	RoomTemp_217: FB_BACnetRM_AI := (Client:=Client,nObjectInstance:=55561);
	TempAdjust_217: FB_BACnetRM_AV := (Client:=Client,nObjectInstance:=55562);
	FilterSign_217: FB_BACnetRM_BI := (Client:=Client,nObjectInstance:=55563);
	FilterSignReset_217: FB_BACnetRM_BV := (Client:=Client,nObjectInstance:=55564);
	RemoteControlStart_217: FB_BACnetRM_BV := (Client:=Client,nObjectInstance:=55565);
	
	RemoteControlTempAdjust_217: FB_BACnetRM_BV := (Client:=Client,nObjectInstance:=55568);
	
	
	
	
	
	
	
	
	
	
	
	
	StartStopCommand_218: FB_BACnetRM_BO := (Client:=Client,nObjectInstance:=55809);
	StartStopStatus_218: FB_BACnetRM_BI := (Client:=Client,nObjectInstance:=55810);
	Alarm_218: FB_BACnetRM_BI := (Client:=Client,nObjectInstance:=55811);
	MalfunctionCode_218: FB_BACnetRM_MI := (Client:=Client,nObjectInstance:=55812);
	
	
	
	
	RoomTemp_218: FB_BACnetRM_AI := (Client:=Client,nObjectInstance:=55817);
	TempAdjust_218: FB_BACnetRM_AV := (Client:=Client,nObjectInstance:=55818);
	FilterSign_218: FB_BACnetRM_BI := (Client:=Client,nObjectInstance:=55819);
	FilterSignReset_218: FB_BACnetRM_BV := (Client:=Client,nObjectInstance:=55820);
	RemoteControlStart_218: FB_BACnetRM_BV := (Client:=Client,nObjectInstance:=55821);
	
	RemoteControlTempAdjust_218: FB_BACnetRM_BV := (Client:=Client,nObjectInstance:=55824);
	
	
	
	
	
	
	
	
	
	
	
	
	StartStopCommand_219: FB_BACnetRM_BO := (Client:=Client,nObjectInstance:=56065);
	StartStopStatus_219: FB_BACnetRM_BI := (Client:=Client,nObjectInstance:=56066);
	Alarm_219: FB_BACnetRM_BI := (Client:=Client,nObjectInstance:=56067);
	MalfunctionCode_219: FB_BACnetRM_MI := (Client:=Client,nObjectInstance:=56068);
	
	
	
	
	RoomTemp_219: FB_BACnetRM_AI := (Client:=Client,nObjectInstance:=56073);
	TempAdjust_219: FB_BACnetRM_AV := (Client:=Client,nObjectInstance:=56074);
	FilterSign_219: FB_BACnetRM_BI := (Client:=Client,nObjectInstance:=56075);
	FilterSignReset_219: FB_BACnetRM_BV := (Client:=Client,nObjectInstance:=56076);
	RemoteControlStart_219: FB_BACnetRM_BV := (Client:=Client,nObjectInstance:=56077);
	
	RemoteControlTempAdjust_219: FB_BACnetRM_BV := (Client:=Client,nObjectInstance:=56080);
	
	
	
	
	
	
	
	
	
	
	
	
	StartStopCommand_220: FB_BACnetRM_BO := (Client:=Client,nObjectInstance:=56321);
	StartStopStatus_220: FB_BACnetRM_BI := (Client:=Client,nObjectInstance:=56322);
	Alarm_220: FB_BACnetRM_BI := (Client:=Client,nObjectInstance:=56323);
	MalfunctionCode_220: FB_BACnetRM_MI := (Client:=Client,nObjectInstance:=56324);
	
	
	
	
	RoomTemp_220: FB_BACnetRM_AI := (Client:=Client,nObjectInstance:=56329);
	TempAdjust_220: FB_BACnetRM_AV := (Client:=Client,nObjectInstance:=56330);
	FilterSign_220: FB_BACnetRM_BI := (Client:=Client,nObjectInstance:=56331);
	FilterSignReset_220: FB_BACnetRM_BV := (Client:=Client,nObjectInstance:=56332);
	RemoteControlStart_220: FB_BACnetRM_BV := (Client:=Client,nObjectInstance:=56333);
	
	RemoteControlTempAdjust_220: FB_BACnetRM_BV := (Client:=Client,nObjectInstance:=56336);
	
	
	
	
	
	
	
	
	
	
	
	
	StartStopCommand_221: FB_BACnetRM_BO := (Client:=Client,nObjectInstance:=56577);
	StartStopStatus_221: FB_BACnetRM_BI := (Client:=Client,nObjectInstance:=56578);
	Alarm_221: FB_BACnetRM_BI := (Client:=Client,nObjectInstance:=56579);
	MalfunctionCode_221: FB_BACnetRM_MI := (Client:=Client,nObjectInstance:=56580);
	
	
	
	
	RoomTemp_221: FB_BACnetRM_AI := (Client:=Client,nObjectInstance:=56585);
	TempAdjust_221: FB_BACnetRM_AV := (Client:=Client,nObjectInstance:=56586);
	FilterSign_221: FB_BACnetRM_BI := (Client:=Client,nObjectInstance:=56587);
	FilterSignReset_221: FB_BACnetRM_BV := (Client:=Client,nObjectInstance:=56588);
	RemoteControlStart_221: FB_BACnetRM_BV := (Client:=Client,nObjectInstance:=56589);
	
	RemoteControlTempAdjust_221: FB_BACnetRM_BV := (Client:=Client,nObjectInstance:=56592);
	
	
	
	
	
	
	
	
	
	
	
	
	StartStopCommand_222: FB_BACnetRM_BO := (Client:=Client,nObjectInstance:=56833);
	StartStopStatus_222: FB_BACnetRM_BI := (Client:=Client,nObjectInstance:=56834);
	Alarm_222: FB_BACnetRM_BI := (Client:=Client,nObjectInstance:=56835);
	MalfunctionCode_222: FB_BACnetRM_MI := (Client:=Client,nObjectInstance:=56836);
	
	
	
	
	RoomTemp_222: FB_BACnetRM_AI := (Client:=Client,nObjectInstance:=56841);
	TempAdjust_222: FB_BACnetRM_AV := (Client:=Client,nObjectInstance:=56842);
	FilterSign_222: FB_BACnetRM_BI := (Client:=Client,nObjectInstance:=56843);
	FilterSignReset_222: FB_BACnetRM_BV := (Client:=Client,nObjectInstance:=56844);
	RemoteControlStart_222: FB_BACnetRM_BV := (Client:=Client,nObjectInstance:=56845);
	
	RemoteControlTempAdjust_222: FB_BACnetRM_BV := (Client:=Client,nObjectInstance:=56848);
	
	
	
	
	
	
	
	
	
	
	
	
	StartStopCommand_223: FB_BACnetRM_BO := (Client:=Client,nObjectInstance:=57089);
	StartStopStatus_223: FB_BACnetRM_BI := (Client:=Client,nObjectInstance:=57090);
	Alarm_223: FB_BACnetRM_BI := (Client:=Client,nObjectInstance:=57091);
	MalfunctionCode_223: FB_BACnetRM_MI := (Client:=Client,nObjectInstance:=57092);
	
	
	
	
	RoomTemp_223: FB_BACnetRM_AI := (Client:=Client,nObjectInstance:=57097);
	TempAdjust_223: FB_BACnetRM_AV := (Client:=Client,nObjectInstance:=57098);
	FilterSign_223: FB_BACnetRM_BI := (Client:=Client,nObjectInstance:=57099);
	FilterSignReset_223: FB_BACnetRM_BV := (Client:=Client,nObjectInstance:=57100);
	RemoteControlStart_223: FB_BACnetRM_BV := (Client:=Client,nObjectInstance:=57101);
	
	RemoteControlTempAdjust_223: FB_BACnetRM_BV := (Client:=Client,nObjectInstance:=57104);
	
	
	
	
	
	
	
	
	
	
	
	
	StartStopCommand_224: FB_BACnetRM_BO := (Client:=Client,nObjectInstance:=57345);
	StartStopStatus_224: FB_BACnetRM_BI := (Client:=Client,nObjectInstance:=57346);
	Alarm_224: FB_BACnetRM_BI := (Client:=Client,nObjectInstance:=57347);
	MalfunctionCode_224: FB_BACnetRM_MI := (Client:=Client,nObjectInstance:=57348);
	
	
	
	
	RoomTemp_224: FB_BACnetRM_AI := (Client:=Client,nObjectInstance:=57353);
	TempAdjust_224: FB_BACnetRM_AV := (Client:=Client,nObjectInstance:=57354);
	FilterSign_224: FB_BACnetRM_BI := (Client:=Client,nObjectInstance:=57355);
	FilterSignReset_224: FB_BACnetRM_BV := (Client:=Client,nObjectInstance:=57356);
	RemoteControlStart_224: FB_BACnetRM_BV := (Client:=Client,nObjectInstance:=57357);
	
	RemoteControlTempAdjust_224: FB_BACnetRM_BV := (Client:=Client,nObjectInstance:=57360);
	
	
	
	
	
	
	
	
	
	
	
	
	StartStopCommand_225: FB_BACnetRM_BO := (Client:=Client,nObjectInstance:=57601);
	StartStopStatus_225: FB_BACnetRM_BI := (Client:=Client,nObjectInstance:=57602);
	Alarm_225: FB_BACnetRM_BI := (Client:=Client,nObjectInstance:=57603);
	MalfunctionCode_225: FB_BACnetRM_MI := (Client:=Client,nObjectInstance:=57604);
	
	
	
	
	RoomTemp_225: FB_BACnetRM_AI := (Client:=Client,nObjectInstance:=57609);
	TempAdjust_225: FB_BACnetRM_AV := (Client:=Client,nObjectInstance:=57610);
	FilterSign_225: FB_BACnetRM_BI := (Client:=Client,nObjectInstance:=57611);
	FilterSignReset_225: FB_BACnetRM_BV := (Client:=Client,nObjectInstance:=57612);
	RemoteControlStart_225: FB_BACnetRM_BV := (Client:=Client,nObjectInstance:=57613);
	
	RemoteControlTempAdjust_225: FB_BACnetRM_BV := (Client:=Client,nObjectInstance:=57616);
	
	
	
	
	
	
	
	
	
	
	
	
	StartStopCommand_226: FB_BACnetRM_BO := (Client:=Client,nObjectInstance:=57857);
	StartStopStatus_226: FB_BACnetRM_BI := (Client:=Client,nObjectInstance:=57858);
	Alarm_226: FB_BACnetRM_BI := (Client:=Client,nObjectInstance:=57859);
	MalfunctionCode_226: FB_BACnetRM_MI := (Client:=Client,nObjectInstance:=57860);
	
	
	
	
	RoomTemp_226: FB_BACnetRM_AI := (Client:=Client,nObjectInstance:=57865);
	TempAdjust_226: FB_BACnetRM_AV := (Client:=Client,nObjectInstance:=57866);
	FilterSign_226: FB_BACnetRM_BI := (Client:=Client,nObjectInstance:=57867);
	FilterSignReset_226: FB_BACnetRM_BV := (Client:=Client,nObjectInstance:=57868);
	RemoteControlStart_226: FB_BACnetRM_BV := (Client:=Client,nObjectInstance:=57869);
	
	RemoteControlTempAdjust_226: FB_BACnetRM_BV := (Client:=Client,nObjectInstance:=57872);
	
	
	
	
	
	
	
	
	
	
	
	
	StartStopCommand_227: FB_BACnetRM_BO := (Client:=Client,nObjectInstance:=58113);
	StartStopStatus_227: FB_BACnetRM_BI := (Client:=Client,nObjectInstance:=58114);
	Alarm_227: FB_BACnetRM_BI := (Client:=Client,nObjectInstance:=58115);
	MalfunctionCode_227: FB_BACnetRM_MI := (Client:=Client,nObjectInstance:=58116);
	
	
	
	
	RoomTemp_227: FB_BACnetRM_AI := (Client:=Client,nObjectInstance:=58121);
	TempAdjust_227: FB_BACnetRM_AV := (Client:=Client,nObjectInstance:=58122);
	FilterSign_227: FB_BACnetRM_BI := (Client:=Client,nObjectInstance:=58123);
	FilterSignReset_227: FB_BACnetRM_BV := (Client:=Client,nObjectInstance:=58124);
	RemoteControlStart_227: FB_BACnetRM_BV := (Client:=Client,nObjectInstance:=58125);
	
	RemoteControlTempAdjust_227: FB_BACnetRM_BV := (Client:=Client,nObjectInstance:=58128);
	
	
	
	
	
	
	
	
	
	
	
	
	StartStopCommand_228: FB_BACnetRM_BO := (Client:=Client,nObjectInstance:=58369);
	StartStopStatus_228: FB_BACnetRM_BI := (Client:=Client,nObjectInstance:=58370);
	Alarm_228: FB_BACnetRM_BI := (Client:=Client,nObjectInstance:=58371);
	MalfunctionCode_228: FB_BACnetRM_MI := (Client:=Client,nObjectInstance:=58372);
	
	
	
	
	RoomTemp_228: FB_BACnetRM_AI := (Client:=Client,nObjectInstance:=58377);
	TempAdjust_228: FB_BACnetRM_AV := (Client:=Client,nObjectInstance:=58378);
	FilterSign_228: FB_BACnetRM_BI := (Client:=Client,nObjectInstance:=58379);
	FilterSignReset_228: FB_BACnetRM_BV := (Client:=Client,nObjectInstance:=58380);
	RemoteControlStart_228: FB_BACnetRM_BV := (Client:=Client,nObjectInstance:=58381);
	
	RemoteControlTempAdjust_228: FB_BACnetRM_BV := (Client:=Client,nObjectInstance:=58384);
	
	
	
	
	
	
	
	
	
	
	
	
	StartStopCommand_229: FB_BACnetRM_BO := (Client:=Client,nObjectInstance:=58625);
	StartStopStatus_229: FB_BACnetRM_BI := (Client:=Client,nObjectInstance:=58626);
	Alarm_229: FB_BACnetRM_BI := (Client:=Client,nObjectInstance:=58627);
	MalfunctionCode_229: FB_BACnetRM_MI := (Client:=Client,nObjectInstance:=58628);
	
	
	
	
	RoomTemp_229: FB_BACnetRM_AI := (Client:=Client,nObjectInstance:=58633);
	TempAdjust_229: FB_BACnetRM_AV := (Client:=Client,nObjectInstance:=58634);
	FilterSign_229: FB_BACnetRM_BI := (Client:=Client,nObjectInstance:=58635);
	FilterSignReset_229: FB_BACnetRM_BV := (Client:=Client,nObjectInstance:=58636);
	RemoteControlStart_229: FB_BACnetRM_BV := (Client:=Client,nObjectInstance:=58637);
	
	RemoteControlTempAdjust_229: FB_BACnetRM_BV := (Client:=Client,nObjectInstance:=58640);
	
	
	
	
	
	
	
	
	
	
	
	
	StartStopCommand_230: FB_BACnetRM_BO := (Client:=Client,nObjectInstance:=58881);
	StartStopStatus_230: FB_BACnetRM_BI := (Client:=Client,nObjectInstance:=58882);
	Alarm_230: FB_BACnetRM_BI := (Client:=Client,nObjectInstance:=58883);
	MalfunctionCode_230: FB_BACnetRM_MI := (Client:=Client,nObjectInstance:=58884);
	
	
	
	
	RoomTemp_230: FB_BACnetRM_AI := (Client:=Client,nObjectInstance:=58889);
	TempAdjust_230: FB_BACnetRM_AV := (Client:=Client,nObjectInstance:=58890);
	FilterSign_230: FB_BACnetRM_BI := (Client:=Client,nObjectInstance:=58891);
	FilterSignReset_230: FB_BACnetRM_BV := (Client:=Client,nObjectInstance:=58892);
	RemoteControlStart_230: FB_BACnetRM_BV := (Client:=Client,nObjectInstance:=58893);
	
	RemoteControlTempAdjust_230: FB_BACnetRM_BV := (Client:=Client,nObjectInstance:=58896);
	
	
	
	
	
	
	
	
	
	
	
	
	StartStopCommand_231: FB_BACnetRM_BO := (Client:=Client,nObjectInstance:=59137);
	StartStopStatus_231: FB_BACnetRM_BI := (Client:=Client,nObjectInstance:=59138);
	Alarm_231: FB_BACnetRM_BI := (Client:=Client,nObjectInstance:=59139);
	MalfunctionCode_231: FB_BACnetRM_MI := (Client:=Client,nObjectInstance:=59140);
	
	
	
	
	RoomTemp_231: FB_BACnetRM_AI := (Client:=Client,nObjectInstance:=59145);
	TempAdjust_231: FB_BACnetRM_AV := (Client:=Client,nObjectInstance:=59146);
	FilterSign_231: FB_BACnetRM_BI := (Client:=Client,nObjectInstance:=59147);
	FilterSignReset_231: FB_BACnetRM_BV := (Client:=Client,nObjectInstance:=59148);
	RemoteControlStart_231: FB_BACnetRM_BV := (Client:=Client,nObjectInstance:=59149);
	
	RemoteControlTempAdjust_231: FB_BACnetRM_BV := (Client:=Client,nObjectInstance:=59152);
	
	
	
	
	
	
	
	
	
	
	
	
	StartStopCommand_232: FB_BACnetRM_BO := (Client:=Client,nObjectInstance:=59393);
	StartStopStatus_232: FB_BACnetRM_BI := (Client:=Client,nObjectInstance:=59394);
	Alarm_232: FB_BACnetRM_BI := (Client:=Client,nObjectInstance:=59395);
	MalfunctionCode_232: FB_BACnetRM_MI := (Client:=Client,nObjectInstance:=59396);
	
	
	
	
	RoomTemp_232: FB_BACnetRM_AI := (Client:=Client,nObjectInstance:=59401);
	TempAdjust_232: FB_BACnetRM_AV := (Client:=Client,nObjectInstance:=59402);
	FilterSign_232: FB_BACnetRM_BI := (Client:=Client,nObjectInstance:=59403);
	FilterSignReset_232: FB_BACnetRM_BV := (Client:=Client,nObjectInstance:=59404);
	RemoteControlStart_232: FB_BACnetRM_BV := (Client:=Client,nObjectInstance:=59405);
	
	RemoteControlTempAdjust_232: FB_BACnetRM_BV := (Client:=Client,nObjectInstance:=59408);
	
	
	
	
	
	
	
	
	
	
	
	
	StartStopCommand_233: FB_BACnetRM_BO := (Client:=Client,nObjectInstance:=59649);
	StartStopStatus_233: FB_BACnetRM_BI := (Client:=Client,nObjectInstance:=59650);
	Alarm_233: FB_BACnetRM_BI := (Client:=Client,nObjectInstance:=59651);
	MalfunctionCode_233: FB_BACnetRM_MI := (Client:=Client,nObjectInstance:=59652);
	
	
	
	
	RoomTemp_233: FB_BACnetRM_AI := (Client:=Client,nObjectInstance:=59657);
	TempAdjust_233: FB_BACnetRM_AV := (Client:=Client,nObjectInstance:=59658);
	FilterSign_233: FB_BACnetRM_BI := (Client:=Client,nObjectInstance:=59659);
	FilterSignReset_233: FB_BACnetRM_BV := (Client:=Client,nObjectInstance:=59660);
	RemoteControlStart_233: FB_BACnetRM_BV := (Client:=Client,nObjectInstance:=59661);
	
	RemoteControlTempAdjust_233: FB_BACnetRM_BV := (Client:=Client,nObjectInstance:=59664);
	
	
	
	
	
	
	
	
	
	
	
	
	StartStopCommand_234: FB_BACnetRM_BO := (Client:=Client,nObjectInstance:=59905);
	StartStopStatus_234: FB_BACnetRM_BI := (Client:=Client,nObjectInstance:=59906);
	Alarm_234: FB_BACnetRM_BI := (Client:=Client,nObjectInstance:=59907);
	MalfunctionCode_234: FB_BACnetRM_MI := (Client:=Client,nObjectInstance:=59908);
	
	
	
	
	RoomTemp_234: FB_BACnetRM_AI := (Client:=Client,nObjectInstance:=59913);
	TempAdjust_234: FB_BACnetRM_AV := (Client:=Client,nObjectInstance:=59914);
	FilterSign_234: FB_BACnetRM_BI := (Client:=Client,nObjectInstance:=59915);
	FilterSignReset_234: FB_BACnetRM_BV := (Client:=Client,nObjectInstance:=59916);
	RemoteControlStart_234: FB_BACnetRM_BV := (Client:=Client,nObjectInstance:=59917);
	
	RemoteControlTempAdjust_234: FB_BACnetRM_BV := (Client:=Client,nObjectInstance:=59920);
	
	
	
	
	
	
	
	
	
	
	
	
	StartStopCommand_235: FB_BACnetRM_BO := (Client:=Client,nObjectInstance:=60161);
	StartStopStatus_235: FB_BACnetRM_BI := (Client:=Client,nObjectInstance:=60162);
	Alarm_235: FB_BACnetRM_BI := (Client:=Client,nObjectInstance:=60163);
	MalfunctionCode_235: FB_BACnetRM_MI := (Client:=Client,nObjectInstance:=60164);
	
	
	
	
	RoomTemp_235: FB_BACnetRM_AI := (Client:=Client,nObjectInstance:=60169);
	TempAdjust_235: FB_BACnetRM_AV := (Client:=Client,nObjectInstance:=60170);
	FilterSign_235: FB_BACnetRM_BI := (Client:=Client,nObjectInstance:=60171);
	FilterSignReset_235: FB_BACnetRM_BV := (Client:=Client,nObjectInstance:=60172);
	RemoteControlStart_235: FB_BACnetRM_BV := (Client:=Client,nObjectInstance:=60173);
	
	RemoteControlTempAdjust_235: FB_BACnetRM_BV := (Client:=Client,nObjectInstance:=60176);
	
	
	
	
	
	
	
	
	
	
	
	
	StartStopCommand_236: FB_BACnetRM_BO := (Client:=Client,nObjectInstance:=60417);
	StartStopStatus_236: FB_BACnetRM_BI := (Client:=Client,nObjectInstance:=60418);
	Alarm_236: FB_BACnetRM_BI := (Client:=Client,nObjectInstance:=60419);
	MalfunctionCode_236: FB_BACnetRM_MI := (Client:=Client,nObjectInstance:=60420);
	
	
	
	
	RoomTemp_236: FB_BACnetRM_AI := (Client:=Client,nObjectInstance:=60425);
	TempAdjust_236: FB_BACnetRM_AV := (Client:=Client,nObjectInstance:=60426);
	FilterSign_236: FB_BACnetRM_BI := (Client:=Client,nObjectInstance:=60427);
	FilterSignReset_236: FB_BACnetRM_BV := (Client:=Client,nObjectInstance:=60428);
	RemoteControlStart_236: FB_BACnetRM_BV := (Client:=Client,nObjectInstance:=60429);
	
	RemoteControlTempAdjust_236: FB_BACnetRM_BV := (Client:=Client,nObjectInstance:=60432);
	
	
	
	
	
	
	
	
	
	
	
	
	StartStopCommand_237: FB_BACnetRM_BO := (Client:=Client,nObjectInstance:=60673);
	StartStopStatus_237: FB_BACnetRM_BI := (Client:=Client,nObjectInstance:=60674);
	Alarm_237: FB_BACnetRM_BI := (Client:=Client,nObjectInstance:=60675);
	MalfunctionCode_237: FB_BACnetRM_MI := (Client:=Client,nObjectInstance:=60676);
	
	
	
	
	RoomTemp_237: FB_BACnetRM_AI := (Client:=Client,nObjectInstance:=60681);
	TempAdjust_237: FB_BACnetRM_AV := (Client:=Client,nObjectInstance:=60682);
	FilterSign_237: FB_BACnetRM_BI := (Client:=Client,nObjectInstance:=60683);
	FilterSignReset_237: FB_BACnetRM_BV := (Client:=Client,nObjectInstance:=60684);
	RemoteControlStart_237: FB_BACnetRM_BV := (Client:=Client,nObjectInstance:=60685);
	
	RemoteControlTempAdjust_237: FB_BACnetRM_BV := (Client:=Client,nObjectInstance:=60688);
	
	
	
	
	
	
	
	
	
	
	
	
	StartStopCommand_238: FB_BACnetRM_BO := (Client:=Client,nObjectInstance:=60929);
	StartStopStatus_238: FB_BACnetRM_BI := (Client:=Client,nObjectInstance:=60930);
	Alarm_238: FB_BACnetRM_BI := (Client:=Client,nObjectInstance:=60931);
	MalfunctionCode_238: FB_BACnetRM_MI := (Client:=Client,nObjectInstance:=60932);
	
	
	
	
	RoomTemp_238: FB_BACnetRM_AI := (Client:=Client,nObjectInstance:=60937);
	TempAdjust_238: FB_BACnetRM_AV := (Client:=Client,nObjectInstance:=60938);
	FilterSign_238: FB_BACnetRM_BI := (Client:=Client,nObjectInstance:=60939);
	FilterSignReset_238: FB_BACnetRM_BV := (Client:=Client,nObjectInstance:=60940);
	RemoteControlStart_238: FB_BACnetRM_BV := (Client:=Client,nObjectInstance:=60941);
	
	RemoteControlTempAdjust_238: FB_BACnetRM_BV := (Client:=Client,nObjectInstance:=60944);
	
	
	
	
	
	
	
	
	
	
	
	
	StartStopCommand_241: FB_BACnetRM_BO := (Client:=Client,nObjectInstance:=61697);
	StartStopStatus_241: FB_BACnetRM_BI := (Client:=Client,nObjectInstance:=61698);
	Alarm_241: FB_BACnetRM_BI := (Client:=Client,nObjectInstance:=61699);
	MalfunctionCode_241: FB_BACnetRM_MI := (Client:=Client,nObjectInstance:=61700);
	
	
	
	
	RoomTemp_241: FB_BACnetRM_AI := (Client:=Client,nObjectInstance:=61705);
	TempAdjust_241: FB_BACnetRM_AV := (Client:=Client,nObjectInstance:=61706);
	FilterSign_241: FB_BACnetRM_BI := (Client:=Client,nObjectInstance:=61707);
	FilterSignReset_241: FB_BACnetRM_BV := (Client:=Client,nObjectInstance:=61708);
	RemoteControlStart_241: FB_BACnetRM_BV := (Client:=Client,nObjectInstance:=61709);
	
	RemoteControlTempAdjust_241: FB_BACnetRM_BV := (Client:=Client,nObjectInstance:=61712);
	
	
	
	
	
	
	
	
	
	
	
	
	StartStopCommand_242: FB_BACnetRM_BO := (Client:=Client,nObjectInstance:=61953);
	StartStopStatus_242: FB_BACnetRM_BI := (Client:=Client,nObjectInstance:=61954);
	Alarm_242: FB_BACnetRM_BI := (Client:=Client,nObjectInstance:=61955);
	MalfunctionCode_242: FB_BACnetRM_MI := (Client:=Client,nObjectInstance:=61956);
	
	
	
	
	RoomTemp_242: FB_BACnetRM_AI := (Client:=Client,nObjectInstance:=61961);
	TempAdjust_242: FB_BACnetRM_AV := (Client:=Client,nObjectInstance:=61962);
	FilterSign_242: FB_BACnetRM_BI := (Client:=Client,nObjectInstance:=61963);
	FilterSignReset_242: FB_BACnetRM_BV := (Client:=Client,nObjectInstance:=61964);
	RemoteControlStart_242: FB_BACnetRM_BV := (Client:=Client,nObjectInstance:=61965);
	
	RemoteControlTempAdjust_242: FB_BACnetRM_BV := (Client:=Client,nObjectInstance:=61968);
	
	
	
	
	
	
	
	
	
	
	
	
	StartStopCommand_243: FB_BACnetRM_BO := (Client:=Client,nObjectInstance:=62209);
	StartStopStatus_243: FB_BACnetRM_BI := (Client:=Client,nObjectInstance:=62210);
	Alarm_243: FB_BACnetRM_BI := (Client:=Client,nObjectInstance:=62211);
	MalfunctionCode_243: FB_BACnetRM_MI := (Client:=Client,nObjectInstance:=62212);
	
	
	
	
	RoomTemp_243: FB_BACnetRM_AI := (Client:=Client,nObjectInstance:=62217);
	TempAdjust_243: FB_BACnetRM_AV := (Client:=Client,nObjectInstance:=62218);
	FilterSign_243: FB_BACnetRM_BI := (Client:=Client,nObjectInstance:=62219);
	FilterSignReset_243: FB_BACnetRM_BV := (Client:=Client,nObjectInstance:=62220);
	RemoteControlStart_243: FB_BACnetRM_BV := (Client:=Client,nObjectInstance:=62221);
	
	RemoteControlTempAdjust_243: FB_BACnetRM_BV := (Client:=Client,nObjectInstance:=62224);
	
	
	
	
	
	
	
	
	
	
	
	
	CL_Rejection_000: FB_BACnetRM_BV := (Client:=Client,nObjectInstance:=17);
	SystemForcedOff_000: FB_BACnetRM_BV := (Client:=Client,nObjectInstance:=21);
	CL_Rejection_064: FB_BACnetRM_BV := (Client:=Client,nObjectInstance:=16401);
	SystemForcedOff_064: FB_BACnetRM_BV := (Client:=Client,nObjectInstance:=16405);
	CL_Rejection_128: FB_BACnetRM_BV := (Client:=Client,nObjectInstance:=32785);
	SystemForcedOff_128: FB_BACnetRM_BV := (Client:=Client,nObjectInstance:=32789);
	CL_Rejection_192: FB_BACnetRM_BV := (Client:=Client,nObjectInstance:=49169);
	SystemForcedOff_192: FB_BACnetRM_BV := (Client:=Client,nObjectInstance:=49173);
END_VAR

Client();
DAIKIN_MasterStation_III_No_10();
StartStopCommand_000();
StartStopStatus_000();
Alarm_000();
MalfunctionCode_000();




RoomTemp_000();
TempAdjust_000();
FilterSign_000();
FilterSignReset_000();
RemoteControlStart_000();

RemoteControlTempAdjust_000();












StartStopCommand_001();
StartStopStatus_001();
Alarm_001();
MalfunctionCode_001();




RoomTemp_001();
TempAdjust_001();
FilterSign_001();
FilterSignReset_001();
RemoteControlStart_001();

RemoteControlTempAdjust_001();












StartStopCommand_002();
StartStopStatus_002();
Alarm_002();
MalfunctionCode_002();




RoomTemp_002();
TempAdjust_002();
FilterSign_002();
FilterSignReset_002();
RemoteControlStart_002();

RemoteControlTempAdjust_002();












StartStopCommand_003();
StartStopStatus_003();
Alarm_003();
MalfunctionCode_003();




RoomTemp_003();
TempAdjust_003();
FilterSign_003();
FilterSignReset_003();
RemoteControlStart_003();

RemoteControlTempAdjust_003();












StartStopCommand_004();
StartStopStatus_004();
Alarm_004();
MalfunctionCode_004();




RoomTemp_004();
TempAdjust_004();
FilterSign_004();
FilterSignReset_004();
RemoteControlStart_004();

RemoteControlTempAdjust_004();












StartStopCommand_005();
StartStopStatus_005();
Alarm_005();
MalfunctionCode_005();




RoomTemp_005();
TempAdjust_005();
FilterSign_005();
FilterSignReset_005();
RemoteControlStart_005();

RemoteControlTempAdjust_005();












StartStopCommand_006();
StartStopStatus_006();
Alarm_006();
MalfunctionCode_006();




RoomTemp_006();
TempAdjust_006();
FilterSign_006();
FilterSignReset_006();
RemoteControlStart_006();

RemoteControlTempAdjust_006();












StartStopCommand_007();
StartStopStatus_007();
Alarm_007();
MalfunctionCode_007();




RoomTemp_007();
TempAdjust_007();
FilterSign_007();
FilterSignReset_007();
RemoteControlStart_007();

RemoteControlTempAdjust_007();












StartStopCommand_008();
StartStopStatus_008();
Alarm_008();
MalfunctionCode_008();




RoomTemp_008();
TempAdjust_008();
FilterSign_008();
FilterSignReset_008();
RemoteControlStart_008();

RemoteControlTempAdjust_008();












StartStopCommand_009();
StartStopStatus_009();
Alarm_009();
MalfunctionCode_009();




RoomTemp_009();
TempAdjust_009();
FilterSign_009();
FilterSignReset_009();
RemoteControlStart_009();

RemoteControlTempAdjust_009();












StartStopCommand_010();
StartStopStatus_010();
Alarm_010();
MalfunctionCode_010();




RoomTemp_010();
TempAdjust_010();
FilterSign_010();
FilterSignReset_010();
RemoteControlStart_010();

RemoteControlTempAdjust_010();












StartStopCommand_011();
StartStopStatus_011();
Alarm_011();
MalfunctionCode_011();




RoomTemp_011();
TempAdjust_011();
FilterSign_011();
FilterSignReset_011();
RemoteControlStart_011();

RemoteControlTempAdjust_011();












StartStopCommand_012();
StartStopStatus_012();
Alarm_012();
MalfunctionCode_012();




RoomTemp_012();
TempAdjust_012();
FilterSign_012();
FilterSignReset_012();
RemoteControlStart_012();

RemoteControlTempAdjust_012();












StartStopCommand_013();
StartStopStatus_013();
Alarm_013();
MalfunctionCode_013();




RoomTemp_013();
TempAdjust_013();
FilterSign_013();
FilterSignReset_013();
RemoteControlStart_013();

RemoteControlTempAdjust_013();












StartStopCommand_014();
StartStopStatus_014();
Alarm_014();
MalfunctionCode_014();




RoomTemp_014();
TempAdjust_014();
FilterSign_014();
FilterSignReset_014();
RemoteControlStart_014();

RemoteControlTempAdjust_014();












StartStopCommand_015();
StartStopStatus_015();
Alarm_015();
MalfunctionCode_015();




RoomTemp_015();
TempAdjust_015();
FilterSign_015();
FilterSignReset_015();
RemoteControlStart_015();

RemoteControlTempAdjust_015();












StartStopCommand_016();
StartStopStatus_016();
Alarm_016();
MalfunctionCode_016();




RoomTemp_016();
TempAdjust_016();
FilterSign_016();
FilterSignReset_016();
RemoteControlStart_016();

RemoteControlTempAdjust_016();












StartStopCommand_017();
StartStopStatus_017();
Alarm_017();
MalfunctionCode_017();




RoomTemp_017();
TempAdjust_017();
FilterSign_017();
FilterSignReset_017();
RemoteControlStart_017();

RemoteControlTempAdjust_017();












StartStopCommand_018();
StartStopStatus_018();
Alarm_018();
MalfunctionCode_018();




RoomTemp_018();
TempAdjust_018();
FilterSign_018();
FilterSignReset_018();
RemoteControlStart_018();

RemoteControlTempAdjust_018();












StartStopCommand_019();
StartStopStatus_019();
Alarm_019();
MalfunctionCode_019();




RoomTemp_019();
TempAdjust_019();
FilterSign_019();
FilterSignReset_019();
RemoteControlStart_019();

RemoteControlTempAdjust_019();












StartStopCommand_020();
StartStopStatus_020();
Alarm_020();
MalfunctionCode_020();




RoomTemp_020();
TempAdjust_020();
FilterSign_020();
FilterSignReset_020();
RemoteControlStart_020();

RemoteControlTempAdjust_020();












StartStopCommand_021();
StartStopStatus_021();
Alarm_021();
MalfunctionCode_021();




RoomTemp_021();
TempAdjust_021();
FilterSign_021();
FilterSignReset_021();
RemoteControlStart_021();

RemoteControlTempAdjust_021();












StartStopCommand_048();
StartStopStatus_048();
Alarm_048();
MalfunctionCode_048();




RoomTemp_048();
TempAdjust_048();
FilterSign_048();
FilterSignReset_048();
RemoteControlStart_048();

RemoteControlTempAdjust_048();












StartStopCommand_049();
StartStopStatus_049();
Alarm_049();
MalfunctionCode_049();




RoomTemp_049();
TempAdjust_049();
FilterSign_049();
FilterSignReset_049();
RemoteControlStart_049();

RemoteControlTempAdjust_049();












StartStopCommand_064();
StartStopStatus_064();
Alarm_064();
MalfunctionCode_064();




RoomTemp_064();
TempAdjust_064();
FilterSign_064();
FilterSignReset_064();
RemoteControlStart_064();

RemoteControlTempAdjust_064();












StartStopCommand_065();
StartStopStatus_065();
Alarm_065();
MalfunctionCode_065();




RoomTemp_065();
TempAdjust_065();
FilterSign_065();
FilterSignReset_065();
RemoteControlStart_065();

RemoteControlTempAdjust_065();












StartStopCommand_066();
StartStopStatus_066();
Alarm_066();
MalfunctionCode_066();




RoomTemp_066();
TempAdjust_066();
FilterSign_066();
FilterSignReset_066();
RemoteControlStart_066();

RemoteControlTempAdjust_066();












StartStopCommand_067();
StartStopStatus_067();
Alarm_067();
MalfunctionCode_067();




RoomTemp_067();
TempAdjust_067();
FilterSign_067();
FilterSignReset_067();
RemoteControlStart_067();

RemoteControlTempAdjust_067();












StartStopCommand_068();
StartStopStatus_068();
Alarm_068();
MalfunctionCode_068();




RoomTemp_068();
TempAdjust_068();
FilterSign_068();
FilterSignReset_068();
RemoteControlStart_068();

RemoteControlTempAdjust_068();












StartStopCommand_069();
StartStopStatus_069();
Alarm_069();
MalfunctionCode_069();




RoomTemp_069();
TempAdjust_069();
FilterSign_069();
FilterSignReset_069();
RemoteControlStart_069();

RemoteControlTempAdjust_069();












StartStopCommand_070();
StartStopStatus_070();
Alarm_070();
MalfunctionCode_070();




RoomTemp_070();
TempAdjust_070();
FilterSign_070();
FilterSignReset_070();
RemoteControlStart_070();

RemoteControlTempAdjust_070();












StartStopCommand_071();
StartStopStatus_071();
Alarm_071();
MalfunctionCode_071();




RoomTemp_071();
TempAdjust_071();
FilterSign_071();
FilterSignReset_071();
RemoteControlStart_071();

RemoteControlTempAdjust_071();












StartStopCommand_072();
StartStopStatus_072();
Alarm_072();
MalfunctionCode_072();




RoomTemp_072();
TempAdjust_072();
FilterSign_072();
FilterSignReset_072();
RemoteControlStart_072();

RemoteControlTempAdjust_072();












StartStopCommand_073();
StartStopStatus_073();
Alarm_073();
MalfunctionCode_073();




RoomTemp_073();
TempAdjust_073();
FilterSign_073();
FilterSignReset_073();
RemoteControlStart_073();

RemoteControlTempAdjust_073();












StartStopCommand_074();
StartStopStatus_074();
Alarm_074();
MalfunctionCode_074();




RoomTemp_074();
TempAdjust_074();
FilterSign_074();
FilterSignReset_074();
RemoteControlStart_074();

RemoteControlTempAdjust_074();












StartStopCommand_075();
StartStopStatus_075();
Alarm_075();
MalfunctionCode_075();




RoomTemp_075();
TempAdjust_075();
FilterSign_075();
FilterSignReset_075();
RemoteControlStart_075();

RemoteControlTempAdjust_075();












StartStopCommand_076();
StartStopStatus_076();
Alarm_076();
MalfunctionCode_076();




RoomTemp_076();
TempAdjust_076();
FilterSign_076();
FilterSignReset_076();
RemoteControlStart_076();

RemoteControlTempAdjust_076();












StartStopCommand_077();
StartStopStatus_077();
Alarm_077();
MalfunctionCode_077();




RoomTemp_077();
TempAdjust_077();
FilterSign_077();
FilterSignReset_077();
RemoteControlStart_077();

RemoteControlTempAdjust_077();












StartStopCommand_078();
StartStopStatus_078();
Alarm_078();
MalfunctionCode_078();




RoomTemp_078();
TempAdjust_078();
FilterSign_078();
FilterSignReset_078();
RemoteControlStart_078();

RemoteControlTempAdjust_078();












StartStopCommand_079();
StartStopStatus_079();
Alarm_079();
MalfunctionCode_079();




RoomTemp_079();
TempAdjust_079();
FilterSign_079();
FilterSignReset_079();
RemoteControlStart_079();

RemoteControlTempAdjust_079();












StartStopCommand_080();
StartStopStatus_080();
Alarm_080();
MalfunctionCode_080();




RoomTemp_080();
TempAdjust_080();
FilterSign_080();
FilterSignReset_080();
RemoteControlStart_080();

RemoteControlTempAdjust_080();












StartStopCommand_081();
StartStopStatus_081();
Alarm_081();
MalfunctionCode_081();




RoomTemp_081();
TempAdjust_081();
FilterSign_081();
FilterSignReset_081();
RemoteControlStart_081();

RemoteControlTempAdjust_081();












StartStopCommand_082();
StartStopStatus_082();
Alarm_082();
MalfunctionCode_082();




RoomTemp_082();
TempAdjust_082();
FilterSign_082();
FilterSignReset_082();
RemoteControlStart_082();

RemoteControlTempAdjust_082();












StartStopCommand_083();
StartStopStatus_083();
Alarm_083();
MalfunctionCode_083();




RoomTemp_083();
TempAdjust_083();
FilterSign_083();
FilterSignReset_083();
RemoteControlStart_083();

RemoteControlTempAdjust_083();












StartStopCommand_084();
StartStopStatus_084();
Alarm_084();
MalfunctionCode_084();




RoomTemp_084();
TempAdjust_084();
FilterSign_084();
FilterSignReset_084();
RemoteControlStart_084();

RemoteControlTempAdjust_084();












StartStopCommand_085();
StartStopStatus_085();
Alarm_085();
MalfunctionCode_085();




RoomTemp_085();
TempAdjust_085();
FilterSign_085();
FilterSignReset_085();
RemoteControlStart_085();

RemoteControlTempAdjust_085();












StartStopCommand_096();
StartStopStatus_096();
Alarm_096();
MalfunctionCode_096();




RoomTemp_096();
TempAdjust_096();
FilterSign_096();
FilterSignReset_096();
RemoteControlStart_096();

RemoteControlTempAdjust_096();












StartStopCommand_097();
StartStopStatus_097();
Alarm_097();
MalfunctionCode_097();




RoomTemp_097();
TempAdjust_097();
FilterSign_097();
FilterSignReset_097();
RemoteControlStart_097();

RemoteControlTempAdjust_097();












StartStopCommand_112();
StartStopStatus_112();
Alarm_112();
MalfunctionCode_112();




RoomTemp_112();
TempAdjust_112();
FilterSign_112();
FilterSignReset_112();
RemoteControlStart_112();

RemoteControlTempAdjust_112();












StartStopCommand_128();
StartStopStatus_128();
Alarm_128();
MalfunctionCode_128();




RoomTemp_128();
TempAdjust_128();
FilterSign_128();
FilterSignReset_128();
RemoteControlStart_128();

RemoteControlTempAdjust_128();












StartStopCommand_129();
StartStopStatus_129();
Alarm_129();
MalfunctionCode_129();




RoomTemp_129();
TempAdjust_129();
FilterSign_129();
FilterSignReset_129();
RemoteControlStart_129();

RemoteControlTempAdjust_129();












StartStopCommand_130();
StartStopStatus_130();
Alarm_130();
MalfunctionCode_130();




RoomTemp_130();
TempAdjust_130();
FilterSign_130();
FilterSignReset_130();
RemoteControlStart_130();

RemoteControlTempAdjust_130();












StartStopCommand_131();
StartStopStatus_131();
Alarm_131();
MalfunctionCode_131();




RoomTemp_131();
TempAdjust_131();
FilterSign_131();
FilterSignReset_131();
RemoteControlStart_131();

RemoteControlTempAdjust_131();












StartStopCommand_132();
StartStopStatus_132();
Alarm_132();
MalfunctionCode_132();




RoomTemp_132();
TempAdjust_132();
FilterSign_132();
FilterSignReset_132();
RemoteControlStart_132();

RemoteControlTempAdjust_132();












StartStopCommand_133();
StartStopStatus_133();
Alarm_133();
MalfunctionCode_133();




RoomTemp_133();
TempAdjust_133();
FilterSign_133();
FilterSignReset_133();
RemoteControlStart_133();

RemoteControlTempAdjust_133();












StartStopCommand_134();
StartStopStatus_134();
Alarm_134();
MalfunctionCode_134();




RoomTemp_134();
TempAdjust_134();
FilterSign_134();
FilterSignReset_134();
RemoteControlStart_134();

RemoteControlTempAdjust_134();












StartStopCommand_135();
StartStopStatus_135();
Alarm_135();
MalfunctionCode_135();




RoomTemp_135();
TempAdjust_135();
FilterSign_135();
FilterSignReset_135();
RemoteControlStart_135();

RemoteControlTempAdjust_135();












StartStopCommand_136();
StartStopStatus_136();
Alarm_136();
MalfunctionCode_136();




RoomTemp_136();
TempAdjust_136();
FilterSign_136();
FilterSignReset_136();
RemoteControlStart_136();

RemoteControlTempAdjust_136();












StartStopCommand_137();
StartStopStatus_137();
Alarm_137();
MalfunctionCode_137();




RoomTemp_137();
TempAdjust_137();
FilterSign_137();
FilterSignReset_137();
RemoteControlStart_137();

RemoteControlTempAdjust_137();












StartStopCommand_138();
StartStopStatus_138();
Alarm_138();
MalfunctionCode_138();




RoomTemp_138();
TempAdjust_138();
FilterSign_138();
FilterSignReset_138();
RemoteControlStart_138();

RemoteControlTempAdjust_138();












StartStopCommand_139();
StartStopStatus_139();
Alarm_139();
MalfunctionCode_139();




RoomTemp_139();
TempAdjust_139();
FilterSign_139();
FilterSignReset_139();
RemoteControlStart_139();

RemoteControlTempAdjust_139();












StartStopCommand_140();
StartStopStatus_140();
Alarm_140();
MalfunctionCode_140();




RoomTemp_140();
TempAdjust_140();
FilterSign_140();
FilterSignReset_140();
RemoteControlStart_140();

RemoteControlTempAdjust_140();












StartStopCommand_141();
StartStopStatus_141();
Alarm_141();
MalfunctionCode_141();




RoomTemp_141();
TempAdjust_141();
FilterSign_141();
FilterSignReset_141();
RemoteControlStart_141();

RemoteControlTempAdjust_141();












StartStopCommand_142();
StartStopStatus_142();
Alarm_142();
MalfunctionCode_142();




RoomTemp_142();
TempAdjust_142();
FilterSign_142();
FilterSignReset_142();
RemoteControlStart_142();

RemoteControlTempAdjust_142();












StartStopCommand_143();
StartStopStatus_143();
Alarm_143();
MalfunctionCode_143();




RoomTemp_143();
TempAdjust_143();
FilterSign_143();
FilterSignReset_143();
RemoteControlStart_143();

RemoteControlTempAdjust_143();












StartStopCommand_144();
StartStopStatus_144();
Alarm_144();
MalfunctionCode_144();




RoomTemp_144();
TempAdjust_144();
FilterSign_144();
FilterSignReset_144();
RemoteControlStart_144();

RemoteControlTempAdjust_144();












StartStopCommand_145();
StartStopStatus_145();
Alarm_145();
MalfunctionCode_145();




RoomTemp_145();
TempAdjust_145();
FilterSign_145();
FilterSignReset_145();
RemoteControlStart_145();

RemoteControlTempAdjust_145();












StartStopCommand_146();
StartStopStatus_146();
Alarm_146();
MalfunctionCode_146();




RoomTemp_146();
TempAdjust_146();
FilterSign_146();
FilterSignReset_146();
RemoteControlStart_146();

RemoteControlTempAdjust_146();












StartStopCommand_147();
StartStopStatus_147();
Alarm_147();
MalfunctionCode_147();




RoomTemp_147();
TempAdjust_147();
FilterSign_147();
FilterSignReset_147();
RemoteControlStart_147();

RemoteControlTempAdjust_147();












StartStopCommand_148();
StartStopStatus_148();
Alarm_148();
MalfunctionCode_148();




RoomTemp_148();
TempAdjust_148();
FilterSign_148();
FilterSignReset_148();
RemoteControlStart_148();

RemoteControlTempAdjust_148();












StartStopCommand_149();
StartStopStatus_149();
Alarm_149();
MalfunctionCode_149();




RoomTemp_149();
TempAdjust_149();
FilterSign_149();
FilterSignReset_149();
RemoteControlStart_149();

RemoteControlTempAdjust_149();












StartStopCommand_150();
StartStopStatus_150();
Alarm_150();
MalfunctionCode_150();




RoomTemp_150();
TempAdjust_150();
FilterSign_150();
FilterSignReset_150();
RemoteControlStart_150();

RemoteControlTempAdjust_150();












StartStopCommand_151();
StartStopStatus_151();
Alarm_151();
MalfunctionCode_151();




RoomTemp_151();
TempAdjust_151();
FilterSign_151();
FilterSignReset_151();
RemoteControlStart_151();

RemoteControlTempAdjust_151();












StartStopCommand_152();
StartStopStatus_152();
Alarm_152();
MalfunctionCode_152();




RoomTemp_152();
TempAdjust_152();
FilterSign_152();
FilterSignReset_152();
RemoteControlStart_152();

RemoteControlTempAdjust_152();












StartStopCommand_153();
StartStopStatus_153();
Alarm_153();
MalfunctionCode_153();




RoomTemp_153();
TempAdjust_153();
FilterSign_153();
FilterSignReset_153();
RemoteControlStart_153();

RemoteControlTempAdjust_153();












StartStopCommand_154();
StartStopStatus_154();
Alarm_154();
MalfunctionCode_154();




RoomTemp_154();
TempAdjust_154();
FilterSign_154();
FilterSignReset_154();
RemoteControlStart_154();

RemoteControlTempAdjust_154();












StartStopCommand_155();
StartStopStatus_155();
Alarm_155();
MalfunctionCode_155();




RoomTemp_155();
TempAdjust_155();
FilterSign_155();
FilterSignReset_155();
RemoteControlStart_155();

RemoteControlTempAdjust_155();












StartStopCommand_156();
StartStopStatus_156();
Alarm_156();
MalfunctionCode_156();




RoomTemp_156();
TempAdjust_156();
FilterSign_156();
FilterSignReset_156();
RemoteControlStart_156();

RemoteControlTempAdjust_156();












StartStopCommand_157();
StartStopStatus_157();
Alarm_157();
MalfunctionCode_157();




RoomTemp_157();
TempAdjust_157();
FilterSign_157();
FilterSignReset_157();
RemoteControlStart_157();

RemoteControlTempAdjust_157();












StartStopCommand_158();
StartStopStatus_158();
Alarm_158();
MalfunctionCode_158();




RoomTemp_158();
TempAdjust_158();
FilterSign_158();
FilterSignReset_158();
RemoteControlStart_158();

RemoteControlTempAdjust_158();












StartStopCommand_159();
StartStopStatus_159();
Alarm_159();
MalfunctionCode_159();




RoomTemp_159();
TempAdjust_159();
FilterSign_159();
FilterSignReset_159();
RemoteControlStart_159();

RemoteControlTempAdjust_159();












StartStopCommand_160();
StartStopStatus_160();
Alarm_160();
MalfunctionCode_160();




RoomTemp_160();
TempAdjust_160();
FilterSign_160();
FilterSignReset_160();
RemoteControlStart_160();

RemoteControlTempAdjust_160();












StartStopCommand_161();
StartStopStatus_161();
Alarm_161();
MalfunctionCode_161();




RoomTemp_161();
TempAdjust_161();
FilterSign_161();
FilterSignReset_161();
RemoteControlStart_161();

RemoteControlTempAdjust_161();












StartStopCommand_162();
StartStopStatus_162();
Alarm_162();
MalfunctionCode_162();




RoomTemp_162();
TempAdjust_162();
FilterSign_162();
FilterSignReset_162();
RemoteControlStart_162();

RemoteControlTempAdjust_162();












StartStopCommand_163();
StartStopStatus_163();
Alarm_163();
MalfunctionCode_163();




RoomTemp_163();
TempAdjust_163();
FilterSign_163();
FilterSignReset_163();
RemoteControlStart_163();

RemoteControlTempAdjust_163();












StartStopCommand_164();
StartStopStatus_164();
Alarm_164();
MalfunctionCode_164();




RoomTemp_164();
TempAdjust_164();
FilterSign_164();
FilterSignReset_164();
RemoteControlStart_164();

RemoteControlTempAdjust_164();












StartStopCommand_165();
StartStopStatus_165();
Alarm_165();
MalfunctionCode_165();




RoomTemp_165();
TempAdjust_165();
FilterSign_165();
FilterSignReset_165();
RemoteControlStart_165();

RemoteControlTempAdjust_165();












StartStopCommand_166();
StartStopStatus_166();
Alarm_166();
MalfunctionCode_166();




RoomTemp_166();
TempAdjust_166();
FilterSign_166();
FilterSignReset_166();
RemoteControlStart_166();

RemoteControlTempAdjust_166();












StartStopCommand_167();
StartStopStatus_167();
Alarm_167();
MalfunctionCode_167();




RoomTemp_167();
TempAdjust_167();
FilterSign_167();
FilterSignReset_167();
RemoteControlStart_167();

RemoteControlTempAdjust_167();












StartStopCommand_168();
StartStopStatus_168();
Alarm_168();
MalfunctionCode_168();




RoomTemp_168();
TempAdjust_168();
FilterSign_168();
FilterSignReset_168();
RemoteControlStart_168();

RemoteControlTempAdjust_168();












StartStopCommand_169();
StartStopStatus_169();
Alarm_169();
MalfunctionCode_169();




RoomTemp_169();
TempAdjust_169();
FilterSign_169();
FilterSignReset_169();
RemoteControlStart_169();

RemoteControlTempAdjust_169();












StartStopCommand_170();
StartStopStatus_170();
Alarm_170();
MalfunctionCode_170();




RoomTemp_170();
TempAdjust_170();
FilterSign_170();
FilterSignReset_170();
RemoteControlStart_170();

RemoteControlTempAdjust_170();












StartStopCommand_171();
StartStopStatus_171();
Alarm_171();
MalfunctionCode_171();




RoomTemp_171();
TempAdjust_171();
FilterSign_171();
FilterSignReset_171();
RemoteControlStart_171();

RemoteControlTempAdjust_171();












StartStopCommand_172();
StartStopStatus_172();
Alarm_172();
MalfunctionCode_172();




RoomTemp_172();
TempAdjust_172();
FilterSign_172();
FilterSignReset_172();
RemoteControlStart_172();

RemoteControlTempAdjust_172();












StartStopCommand_173();
StartStopStatus_173();
Alarm_173();
MalfunctionCode_173();




RoomTemp_173();
TempAdjust_173();
FilterSign_173();
FilterSignReset_173();
RemoteControlStart_173();

RemoteControlTempAdjust_173();












StartStopCommand_192();
StartStopStatus_192();
Alarm_192();
MalfunctionCode_192();




RoomTemp_192();
TempAdjust_192();
FilterSign_192();
FilterSignReset_192();
RemoteControlStart_192();

RemoteControlTempAdjust_192();












StartStopCommand_193();
StartStopStatus_193();
Alarm_193();
MalfunctionCode_193();




RoomTemp_193();
TempAdjust_193();
FilterSign_193();
FilterSignReset_193();
RemoteControlStart_193();

RemoteControlTempAdjust_193();












StartStopCommand_194();
StartStopStatus_194();
Alarm_194();
MalfunctionCode_194();




RoomTemp_194();
TempAdjust_194();
FilterSign_194();
FilterSignReset_194();
RemoteControlStart_194();

RemoteControlTempAdjust_194();












StartStopCommand_195();
StartStopStatus_195();
Alarm_195();
MalfunctionCode_195();




RoomTemp_195();
TempAdjust_195();
FilterSign_195();
FilterSignReset_195();
RemoteControlStart_195();

RemoteControlTempAdjust_195();












StartStopCommand_196();
StartStopStatus_196();
Alarm_196();
MalfunctionCode_196();




RoomTemp_196();
TempAdjust_196();
FilterSign_196();
FilterSignReset_196();
RemoteControlStart_196();

RemoteControlTempAdjust_196();












StartStopCommand_197();
StartStopStatus_197();
Alarm_197();
MalfunctionCode_197();




RoomTemp_197();
TempAdjust_197();
FilterSign_197();
FilterSignReset_197();
RemoteControlStart_197();

RemoteControlTempAdjust_197();












StartStopCommand_198();
StartStopStatus_198();
Alarm_198();
MalfunctionCode_198();




RoomTemp_198();
TempAdjust_198();
FilterSign_198();
FilterSignReset_198();
RemoteControlStart_198();

RemoteControlTempAdjust_198();












StartStopCommand_199();
StartStopStatus_199();
Alarm_199();
MalfunctionCode_199();




RoomTemp_199();
TempAdjust_199();
FilterSign_199();
FilterSignReset_199();
RemoteControlStart_199();

RemoteControlTempAdjust_199();












//StartStopCommand_200();
//StartStopStatus_200();
//Alarm_200();
//MalfunctionCode_200();




//RoomTemp_200();
//TempAdjust_200();
//FilterSign_200();
//FilterSignReset_200();
//RemoteControlStart_200();
//
//RemoteControlTempAdjust_200();

//










StartStopCommand_201();
StartStopStatus_201();
Alarm_201();
MalfunctionCode_201();




RoomTemp_201();
TempAdjust_201();
FilterSign_201();
FilterSignReset_201();
RemoteControlStart_201();

RemoteControlTempAdjust_201();












StartStopCommand_202();
StartStopStatus_202();
Alarm_202();
MalfunctionCode_202();




RoomTemp_202();
TempAdjust_202();
FilterSign_202();
FilterSignReset_202();
RemoteControlStart_202();

RemoteControlTempAdjust_202();












StartStopCommand_203();
StartStopStatus_203();
Alarm_203();
MalfunctionCode_203();




RoomTemp_203();
TempAdjust_203();
FilterSign_203();
FilterSignReset_203();
RemoteControlStart_203();

RemoteControlTempAdjust_203();












StartStopCommand_204();
StartStopStatus_204();
Alarm_204();
MalfunctionCode_204();




RoomTemp_204();
TempAdjust_204();
FilterSign_204();
FilterSignReset_204();
RemoteControlStart_204();

RemoteControlTempAdjust_204();












StartStopCommand_205();
StartStopStatus_205();
Alarm_205();
MalfunctionCode_205();




RoomTemp_205();
TempAdjust_205();
FilterSign_205();
FilterSignReset_205();
RemoteControlStart_205();

RemoteControlTempAdjust_205();












StartStopCommand_206();
StartStopStatus_206();
Alarm_206();
MalfunctionCode_206();




RoomTemp_206();
TempAdjust_206();
FilterSign_206();
FilterSignReset_206();
RemoteControlStart_206();

RemoteControlTempAdjust_206();












StartStopCommand_207();
StartStopStatus_207();
Alarm_207();
MalfunctionCode_207();




RoomTemp_207();
TempAdjust_207();
FilterSign_207();
FilterSignReset_207();
RemoteControlStart_207();

RemoteControlTempAdjust_207();












StartStopCommand_208();
StartStopStatus_208();
Alarm_208();
MalfunctionCode_208();




RoomTemp_208();
TempAdjust_208();
FilterSign_208();
FilterSignReset_208();
RemoteControlStart_208();

RemoteControlTempAdjust_208();












StartStopCommand_209();
StartStopStatus_209();
Alarm_209();
MalfunctionCode_209();




RoomTemp_209();
TempAdjust_209();
FilterSign_209();
FilterSignReset_209();
RemoteControlStart_209();

RemoteControlTempAdjust_209();












StartStopCommand_210();
StartStopStatus_210();
Alarm_210();
MalfunctionCode_210();




RoomTemp_210();
TempAdjust_210();
FilterSign_210();
FilterSignReset_210();
RemoteControlStart_210();

RemoteControlTempAdjust_210();












StartStopCommand_211();
StartStopStatus_211();
Alarm_211();
MalfunctionCode_211();




RoomTemp_211();
TempAdjust_211();
FilterSign_211();
FilterSignReset_211();
RemoteControlStart_211();

RemoteControlTempAdjust_211();












StartStopCommand_212();
StartStopStatus_212();
Alarm_212();
MalfunctionCode_212();




RoomTemp_212();
TempAdjust_212();
FilterSign_212();
FilterSignReset_212();
RemoteControlStart_212();

RemoteControlTempAdjust_212();












StartStopCommand_213();
StartStopStatus_213();
Alarm_213();
MalfunctionCode_213();




RoomTemp_213();
TempAdjust_213();
FilterSign_213();
FilterSignReset_213();
RemoteControlStart_213();

RemoteControlTempAdjust_213();












StartStopCommand_214();
StartStopStatus_214();
Alarm_214();
MalfunctionCode_214();




RoomTemp_214();
TempAdjust_214();
FilterSign_214();
FilterSignReset_214();
RemoteControlStart_214();

RemoteControlTempAdjust_214();












StartStopCommand_215();
StartStopStatus_215();
Alarm_215();
MalfunctionCode_215();




RoomTemp_215();
TempAdjust_215();
FilterSign_215();
FilterSignReset_215();
RemoteControlStart_215();

RemoteControlTempAdjust_215();












StartStopCommand_216();
StartStopStatus_216();
Alarm_216();
MalfunctionCode_216();




RoomTemp_216();
TempAdjust_216();
FilterSign_216();
FilterSignReset_216();
RemoteControlStart_216();

RemoteControlTempAdjust_216();












StartStopCommand_217();
StartStopStatus_217();
Alarm_217();
MalfunctionCode_217();




RoomTemp_217();
TempAdjust_217();
FilterSign_217();
FilterSignReset_217();
RemoteControlStart_217();

RemoteControlTempAdjust_217();












StartStopCommand_218();
StartStopStatus_218();
Alarm_218();
MalfunctionCode_218();




RoomTemp_218();
TempAdjust_218();
FilterSign_218();
FilterSignReset_218();
RemoteControlStart_218();

RemoteControlTempAdjust_218();












StartStopCommand_219();
StartStopStatus_219();
Alarm_219();
MalfunctionCode_219();




RoomTemp_219();
TempAdjust_219();
FilterSign_219();
FilterSignReset_219();
RemoteControlStart_219();

RemoteControlTempAdjust_219();












StartStopCommand_220();
StartStopStatus_220();
Alarm_220();
MalfunctionCode_220();




RoomTemp_220();
TempAdjust_220();
FilterSign_220();
FilterSignReset_220();
RemoteControlStart_220();

RemoteControlTempAdjust_220();












StartStopCommand_221();
StartStopStatus_221();
Alarm_221();
MalfunctionCode_221();




RoomTemp_221();
TempAdjust_221();
FilterSign_221();
FilterSignReset_221();
RemoteControlStart_221();

RemoteControlTempAdjust_221();












StartStopCommand_222();
StartStopStatus_222();
Alarm_222();
MalfunctionCode_222();




RoomTemp_222();
TempAdjust_222();
FilterSign_222();
FilterSignReset_222();
RemoteControlStart_222();

RemoteControlTempAdjust_222();












StartStopCommand_223();
StartStopStatus_223();
Alarm_223();
MalfunctionCode_223();




RoomTemp_223();
TempAdjust_223();
FilterSign_223();
FilterSignReset_223();
RemoteControlStart_223();

RemoteControlTempAdjust_223();












StartStopCommand_224();
StartStopStatus_224();
Alarm_224();
MalfunctionCode_224();




RoomTemp_224();
TempAdjust_224();
FilterSign_224();
FilterSignReset_224();
RemoteControlStart_224();

RemoteControlTempAdjust_224();












StartStopCommand_225();
StartStopStatus_225();
Alarm_225();
MalfunctionCode_225();




RoomTemp_225();
TempAdjust_225();
FilterSign_225();
FilterSignReset_225();
RemoteControlStart_225();

RemoteControlTempAdjust_225();












StartStopCommand_226();
StartStopStatus_226();
Alarm_226();
MalfunctionCode_226();




RoomTemp_226();
TempAdjust_226();
FilterSign_226();
FilterSignReset_226();
RemoteControlStart_226();

RemoteControlTempAdjust_226();












StartStopCommand_227();
StartStopStatus_227();
Alarm_227();
MalfunctionCode_227();




RoomTemp_227();
TempAdjust_227();
FilterSign_227();
FilterSignReset_227();
RemoteControlStart_227();

RemoteControlTempAdjust_227();












StartStopCommand_228();
StartStopStatus_228();
Alarm_228();
MalfunctionCode_228();




RoomTemp_228();
TempAdjust_228();
FilterSign_228();
FilterSignReset_228();
RemoteControlStart_228();

RemoteControlTempAdjust_228();












StartStopCommand_229();
StartStopStatus_229();
Alarm_229();
MalfunctionCode_229();




RoomTemp_229();
TempAdjust_229();
FilterSign_229();
FilterSignReset_229();
RemoteControlStart_229();

RemoteControlTempAdjust_229();












StartStopCommand_230();
StartStopStatus_230();
Alarm_230();
MalfunctionCode_230();




RoomTemp_230();
TempAdjust_230();
FilterSign_230();
FilterSignReset_230();
RemoteControlStart_230();

RemoteControlTempAdjust_230();












StartStopCommand_231();
StartStopStatus_231();
Alarm_231();
MalfunctionCode_231();




RoomTemp_231();
TempAdjust_231();
FilterSign_231();
FilterSignReset_231();
RemoteControlStart_231();

RemoteControlTempAdjust_231();












StartStopCommand_232();
StartStopStatus_232();
Alarm_232();
MalfunctionCode_232();




RoomTemp_232();
TempAdjust_232();
FilterSign_232();
FilterSignReset_232();
RemoteControlStart_232();

RemoteControlTempAdjust_232();












StartStopCommand_233();
StartStopStatus_233();
Alarm_233();
MalfunctionCode_233();




RoomTemp_233();
TempAdjust_233();
FilterSign_233();
FilterSignReset_233();
RemoteControlStart_233();

RemoteControlTempAdjust_233();












StartStopCommand_234();
StartStopStatus_234();
Alarm_234();
MalfunctionCode_234();




RoomTemp_234();
TempAdjust_234();
FilterSign_234();
FilterSignReset_234();
RemoteControlStart_234();

RemoteControlTempAdjust_234();












StartStopCommand_235();
StartStopStatus_235();
Alarm_235();
MalfunctionCode_235();




RoomTemp_235();
TempAdjust_235();
FilterSign_235();
FilterSignReset_235();
RemoteControlStart_235();

RemoteControlTempAdjust_235();












StartStopCommand_236();
StartStopStatus_236();
Alarm_236();
MalfunctionCode_236();




RoomTemp_236();
TempAdjust_236();
FilterSign_236();
FilterSignReset_236();
RemoteControlStart_236();

RemoteControlTempAdjust_236();












StartStopCommand_237();
StartStopStatus_237();
Alarm_237();
MalfunctionCode_237();




RoomTemp_237();
TempAdjust_237();
FilterSign_237();
FilterSignReset_237();
RemoteControlStart_237();

RemoteControlTempAdjust_237();












StartStopCommand_238();
StartStopStatus_238();
Alarm_238();
MalfunctionCode_238();




RoomTemp_238();
TempAdjust_238();
FilterSign_238();
FilterSignReset_238();
RemoteControlStart_238();

RemoteControlTempAdjust_238();












StartStopCommand_241();
StartStopStatus_241();
Alarm_241();
MalfunctionCode_241();




RoomTemp_241();
TempAdjust_241();
FilterSign_241();
FilterSignReset_241();
RemoteControlStart_241();

RemoteControlTempAdjust_241();












StartStopCommand_242();
StartStopStatus_242();
Alarm_242();
MalfunctionCode_242();




RoomTemp_242();
TempAdjust_242();
FilterSign_242();
FilterSignReset_242();
RemoteControlStart_242();

RemoteControlTempAdjust_242();












StartStopCommand_243();
StartStopStatus_243();
Alarm_243();
MalfunctionCode_243();




RoomTemp_243();
TempAdjust_243();
FilterSign_243();
FilterSignReset_243();
RemoteControlStart_243();

RemoteControlTempAdjust_243();












CL_Rejection_000();
SystemForcedOff_000();
CL_Rejection_064();
SystemForcedOff_064();
CL_Rejection_128();
SystemForcedOff_128();
CL_Rejection_192();
SystemForcedOff_192();

END_FUNCTION_BLOCK

(* stored: Version 1.1.0.1, ProductVersion 3.1.4024.14
   POU FB_BACnet_DAIKIN_MasterStation_III_No_10: Id {3918e4d6-2e08-41fb-977c-1d1d550de316}, SpecialFunc None *)
